SUBAPPLICATION AX_AND_2_DUAL (* Gated Heben/Senken-Paar mit gemeinsamer Freigabe: OUT_UP = IN_UP AND IN_PERMIT, OUT_DOWN = IN_DOWN AND IN_PERMIT, OUT_PERMIT = IN_PERMIT durchgereicht (fuer einen dritten Verbraucher, der die rohe Freigabe selbst braucht - z.B. eine Statusanzeige). Spart 2x AX_AND_2 + 1x AX_SPLIT_3 als Einzelbausteine, wo immer ein Heben/Senken-Signalpaar dieselbe Freigabe gegatet braucht. *)
  (* Standard: 61499-2; Description: Copyright (c) 2026 Meisterschulen am Ostbahnhof This program and the accompanying materials are made available under the terms of the Eclipse Public License 2.0 which is available at https://www.eclipse.org/legal/epl-2.0/ SPDX-License-Identifier: EPL-2.0 *)
  (* Version 1.0, 2026-09-27, Franz Höpfinger, Meisterschulen am Ostbahnhof, initial implementation - generische Gate-Kombination fuer ein Heben/Senken-Signalpaar mit gemeinsamer Freigabe, IN_PERMIT zusaetzlich unveraendert als OUT_PERMIT durchgereicht. *)
  PACKAGE MyLib::sys;
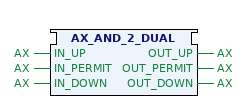
  SOCKETS
    IN_UP : adapter::types::unidirectional::AX; (* Rohes Heben-Signal, wird mit IN_PERMIT gegated *)
    IN_PERMIT : adapter::types::unidirectional::AX; (* Gemeinsame Freigabe fuer IN_UP/IN_DOWN, zusaetzlich unveraendert an OUT_PERMIT durchgereicht *)
    IN_DOWN : adapter::types::unidirectional::AX; (* Rohes Senken-Signal, wird mit IN_PERMIT gegated *)
  END_SOCKETS
  PLUGS
    OUT_UP : adapter::types::unidirectional::AX; (* IN_UP AND IN_PERMIT *)
    OUT_PERMIT : adapter::types::unidirectional::AX; (* IN_PERMIT unveraendert durchgereicht (fuer einen dritten Verbraucher, z.B. eine Statusanzeige) *)
    OUT_DOWN : adapter::types::unidirectional::AX; (* IN_DOWN AND IN_PERMIT *)
  END_PLUGS
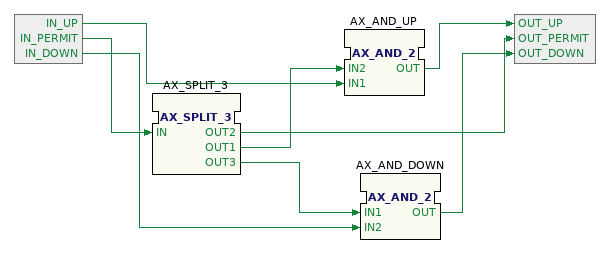
  FBS
    AX_AND_UP : adapter::booleanOperators::AX_AND_2;
    AX_AND_DOWN : adapter::booleanOperators::AX_AND_2;
    AX_SPLIT_3 : adapter::events::unidirectional::AX_SPLIT_3;
  END_FBS
  ADAPTER_CONNECTIONS
    AX_AND_UP.OUT TO OUT_UP;
    AX_AND_DOWN.OUT TO OUT_DOWN;
    IN_PERMIT TO AX_SPLIT_3.IN;
    AX_SPLIT_3.OUT2 TO OUT_PERMIT;
    AX_SPLIT_3.OUT1 TO AX_AND_UP.IN2;
    AX_SPLIT_3.OUT3 TO AX_AND_DOWN.IN1;
    IN_DOWN TO AX_AND_DOWN.IN2;
    IN_UP TO AX_AND_UP.IN1;
  END_CONNECTIONS
END_SUBAPPLICATION
